{attribute addProperty BoxType "EP7402-0057-0017"}
{attribute addProperty Id "StatusAT %I*Status_26CB4AD2162"}
{attribute addProperty CRC "1223458837"}
{attribute addProperty SizeInBites "16"}
{attribute addProperty SizeInBytes "2"}
TYPE STM_Status_Channel_48EC8015 :
STRUCT
	{attribute addProperty Name "Status"}
	Status AT %I* : Status_26CB4AD2;
END_STRUCT
END_TYPE

(* stored: Version 1.2.0.0, ProductVersion 3.1.4024.9
   DUT STM_Status_Channel_48EC8015: Id {ac86330b-73c0-4af6-b822-4da020d52cdb} *)
